ABB RobotStudio station: MiniProiect_v2final.rspag

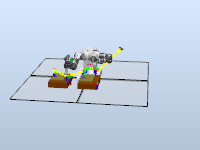
--- station ---
Station MiniProiect2 (saved by RobotStudio 7.0.8730.594)
Controller YuMi
  mechanical unit ROB_R: IRB14000_0.5_0.5_R, 6 joints, base frame (0, 0, 0) mm
  mechanical unit ROB_R_7: IRB14000_0.5_0.5_R, 1 joints, base frame (0, 0, 0) mm
  mechanical unit ROB_L: IRB14000_0.5_0.5_L, 6 joints, base frame (0, 0, 0) mm
  mechanical unit ROB_L_7: IRB14000_0.5_0.5_L, 1 joints, base frame (0, 0, 0) mm
Layout (positions relative to the parent item):
  - IRB14000_0.5_0.5 [mechanism, from Robots\IRB14000_0.5_0.5__01.rslib] at (0, 0, 0) mm
  - IRB14000_0.5_0.5_R [mechanism, from Robots\IRB14000_0.5_0.5__01.rslib] at (0, 0, 0) mm; joint values [2.2467, -1.1641, -0.2452, 0.0995, -2.8474, 1.8685, 0.012] (rad or m)
  - IRB14000_0.5_0.5_L [mechanism, from Robots\IRB14000_0.5_0.5__01.rslib] at (0, 0, 0) mm; joint values [-0.9882, -1.1775, 0.9709, 1.2171, -1.1721, -1.5184, 1.7927] (rad or m)
  - Curve_thing [part, from Training Objects\Curve_Thing.rslib] at (300, -50, 90) mm
  - Smart_Gripper_Servo_Fingers [mechanism, from Tools\ABB_Smart_Gripper_Servo_Fingers.rslib] at (305.45, 153.32, 394.2) mm, rotated rx 180 ry 0 rz 180 deg; joint values [0] (rad or m)
  - MyTool_2 [mechanism, from Training Objects\myTool.rslib] at (623.67, -200, 500.53) mm, rotated rx -180 ry 38 rz -180 deg
  - Curve [part, from Training Objects\Curve_Thing.rslib] at (300, -500, 90) mm
  - Part_3 [part] at (500.36, 1.06, 247.73) mm, rotated rx 179.59 ry 1.47 rz 162.83 deg
  - Part_4 [part] at (500, 0, 250) mm, rotated rx 180 ry 0 rz 84.95 deg
  - Attacher [smart component, from Components\Attacher.rslib]
      properties: Parent=MyTool_2; Flange=0; Child=Part_3; Mount=false; Offset=[0 0 0]; Orientation=[0 0 0]
  - Detacher [smart component, from Components\Detacher.rslib]
      properties: Child=Part_3; KeepPosition=true
  - CollisionSensor [smart component, from Components\CollisionSensor.rslib]
      properties: Object1=MyTool_2; Object2=Part_3; NearMiss=0.01; Part1=(none); Part2=(none); CollisionType=0
    - _sensorPart_ [part]
  - CollisionSensor_2 [smart component, from Components\CollisionSensor.rslib]
      properties: Object1=MyTool_2; Object2=Part_4; NearMiss=0.01; Part1=(none); Part2=(none); CollisionType=0
    - _sensorPart_ [part]
  - Positioner [smart component, from Components\Positioner.rslib]
      properties: Object=Part_3; Position=[0.477076 -0.45939 0.25]; Orientation=[0 0 0]; Reference=Global; ReferenceObject=(none)
Attachment: Smart_Gripper_Servo_Fingers is attached to IRB14000_0.5_0.5_L / Link7
Attachment: MyTool_2 is attached to IRB14000_0.5_0.5_R / Link7
Station signals: DI reset
Station logic (signal -> signal, property => property):
  MiniProiect2.reset -> Positioner.Execute
  CollisionSensor.SensorOut -> Attacher.Execute
  CollisionSensor_2.SensorOut -> Detacher.Execute

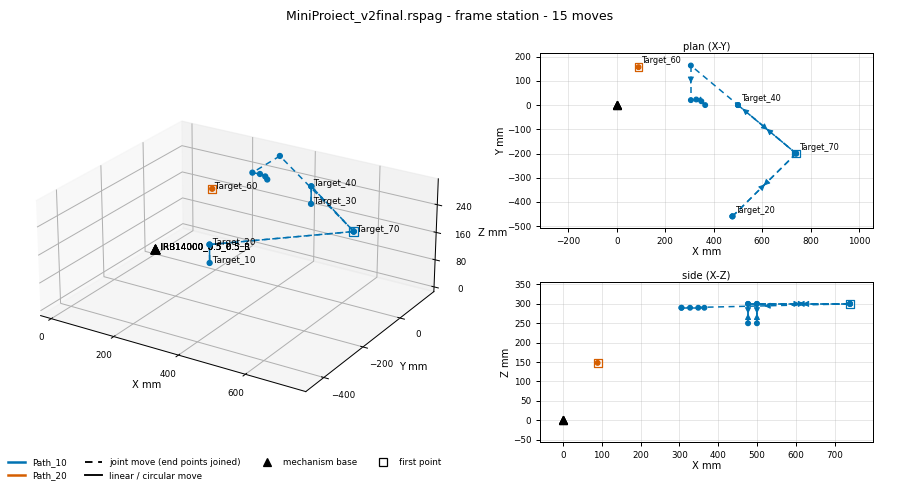
[picture p0: tool path of MiniProiect_v2final.rspag in frame station, 15 of 27 moves have a stored position in this frame; points joined in program order, loops and branches not executed]
--- Backups/YuMi/RAPID/TASK1/PROGMOD/CalibData.mod ---
MODULE CalibData
	PERS tooldata IRB5350_Gripper:=[TRUE,[[350,0,243],[0,1,0,0]],[1,[0,0,100],[1,0,0,0],0,0,0]];
	PERS tooldata MyTool:=[TRUE,[[31.7926,0,229.639],[0.945519,0,0.325568,0]],[1,[0,0,1],[1,0,0,0],0,0,0]];
ENDMODULE

--- Backups/YuMi/RAPID/TASK1/PROGMOD/Module1.mod ---
MODULE Module1
	CONST robtarget Target_70:=[[740,-200.004,300],[0,0,1,0],[1,-1,0,4],[-101.764306343,9E+09,9E+09,9E+09,9E+09,9E+09]];
	CONST robtarget Target_10:=[[477.07615446,-459.390112623,249.999908006],[-0.000000218,0.173648122,0.984807763,-0.000000081],[1,-2,0,4],[-101.764290321,9E+09,9E+09,9E+09,9E+09,9E+09]];
	CONST robtarget Target_20:=[[477.076,-459.39,300],[0,0.173648178,0.984807753,0],[1,-2,0,4],[-101.764306343,9E+09,9E+09,9E+09,9E+09,9E+09]];
	CONST robtarget Target_40:=[[500,0,300],[0,-0.173648177,0.984807753,0],[1,-2,0,4],[-101.764306343,9E+09,9E+09,9E+09,9E+09,9E+09]];
	CONST robtarget Target_30:=[[500,0,250],[0,-0.173648177,0.984807753,0],[1,-2,0,4],[-101.764306343,9E+09,9E+09,9E+09,9E+09,9E+09]];
    !***********************************************************
    !
    ! Module:  Module1
    !
    ! Description:
    !   <Insert description here>
    !
    ! Author: theod
    !
    ! Version: 1.0
    !
    !***********************************************************


    !***********************************************************
    !
    ! Procedure main
    !
    !   This is the entry point of your program
    !
    !***********************************************************
    PROC main()
        !Add your code here
    ENDPROC
	PROC Path_10()
	    MoveJ Target_70,v200,fine,MyTool\WObj:=wobj0;
	    MoveJ Target_20,v200,fine,MyTool\WObj:=wobj0;
	    MoveJ Target_10,v200,fine,MyTool\WObj:=wobj0;
	    MoveL Target_20,v1000,z100,MyTool\WObj:=wobj0;
	    MoveJ Target_70,v200,fine,MyTool\WObj:=wobj0;
	    MoveJ Target_40,v200,fine,MyTool\WObj:=wobj0;
	    MoveJ Target_30,v200,fine,MyTool\WObj:=wobj0;
	    MoveL Target_40,v1000,z100,MyTool\WObj:=wobj0;
	    MoveJ Target_70,v200,fine,MyTool\WObj:=wobj0;
	ENDPROC
ENDMODULE

--- Backups/YuMi/RAPID/TASK2/PROGMOD/CalibData.mod ---
MODULE CalibData
	PERS wobjdata Workobject_2:=[FALSE,TRUE,"",[[521.091,38.6689,180],[0,0.737574,0.675266,0]],[[0,0,0],[1,0,0,0]]];
	PERS wobjdata Workobject_3:=[FALSE,TRUE,"",[[477.076,-459.39,180],[0,0.737574,0.675266,0]],[[0,0,0],[1,0,0,0]]];
ENDMODULE

--- Backups/YuMi/RAPID/TASK2/PROGMOD/Module1.mod ---
MODULE Module1
	PERS tooldata Servo:=[TRUE,[[0,0,114.2],[1,0,0,0]],[0.215,[8.7,12.3,49.2],[1,0,0,0],0.00021,0.00024,0.00009]];
	PERS wobjdata Workobject_1:=[FALSE,TRUE,"",[[699.999,249.996,180],[0,-0.707107,0.707107,0]],[[0,0,0],[1,0,0,0]]];
	CONST robtarget Target_10:=[[86.674039551,394.552253174,-110],[0.707106781,0,0,0.707106781],[-1,-1,1,5],[135,9E+09,9E+09,9E+09,9E+09,9E+09]];
	CONST robtarget Target_20:=[[229.547583792,394.552253174,-110],[0.707106781,0,0,0.707106781],[-1,-1,1,5],[135,9E+09,9E+09,9E+09,9E+09,9E+09]];
	CONST robtarget Target_30:=[[226.937896068,372.374442925,-110],[0.707106781,0,0,0.707106781],[-1,-1,1,5],[135,9E+09,9E+09,9E+09,9E+09,9E+09]];
	CONST robtarget Target_40:=[[234.243334971,351.272398004,-110],[0.707106781,0,0,0.707106781],[-1,-1,1,5],[135,9E+09,9E+09,9E+09,9E+09,9E+09]];
	CONST robtarget Target_50:=[[250.00671167,335.455265126,-110],[0.707106781,0,0,0.707106781],[-1,-1,1,5],[135,9E+09,9E+09,9E+09,9E+09,9E+09]];
	CONST robtarget Target_60:=[[93.373882043,610.611053577,32.086529783],[0.674322362,0.323188765,0.416542029,-0.517040725],[0,0,0,4],[101.964427132,9E+09,9E+09,9E+09,9E+09,9E+09]];
	CONST jointtarget JointTarget_1:=[[-32.11,-102,-5.71,-103,-56.09,83.99],[0,9E+09,9E+09,9E+09,9E+09,9E+09]];
    CONST jointtarget JointTarget_2:=[[-32.11,-48.5,-5.71,-103,-56.09,83.99],[0,9E+09,9E+09,9E+09,9E+09,9E+09]];

    PROC main()
        !Path_Shake;
        userCommand;
    ENDPROC
	PROC Path_10()
	    MoveJ Target_10,v300,fine,Servo\WObj:=Workobject_1;
	    MoveJ Target_20,v300,fine,Servo\WObj:=Workobject_1;
	    MoveJ Target_30,v300,fine,Servo\WObj:=Workobject_1;
	    MoveJ Target_40,v300,fine,Servo\WObj:=Workobject_1;
	    MoveJ Target_50,v300,fine,Servo\WObj:=Workobject_1;
	ENDPROC
	PROC Path_20()
	    MoveJ Target_60,v300,fine,Servo\WObj:=Workobject_1;
	    MoveAbsJ JointTarget_1,v300,fine,Servo\WObj:=Workobject_1;
	ENDPROC

    PROC userCommand()
        VAR num valTranslare;
        CONST robtarget Target_70:=[[96.674039551,394.552253174,-110],[0.707106781,0,0,0.707106781],[-1,-1,1,5],[135,9E+09,9E+09,9E+09,9E+09,9E+09]];
        CONST robtarget Target_80:=[[126.674039551,394.552253174,-110],[0.707106781,0,0,0.707106781],[-1,-1,1,5],[135,9E+09,9E+09,9E+09,9E+09,9E+09]];
        CONST robtarget Target_90:=[[126.674039551,394.552253174,-90],[0.707106781,0,0,0.707106781],[-1,-1,1,5],[135,9E+09,9E+09,9E+09,9E+09,9E+09]];
        CONST robtarget Target_100:=[[96.674039551,394.552253174,-90],[0.707106781,0,0,0.707106781],[-1,-1,1,5],[135,9E+09,9E+09,9E+09,9E+09,9E+09]];
        TPReadNum valTranslare,"Dati o vloare pt translarea pe Z:";
        MoveJ RelTool(Target_10,0,0,valTranslare),v300,fine,Servo\WObj:=Workobject_1;
        WaitTime 2;
        MoveJ RelTool(Target_70,0,0,valTranslare),v300,fine,Servo\WObj:=Workobject_1;
        WaitTime 2;
        MoveJ RelTool(Target_80,0,0,valTranslare),v300,fine,Servo\WObj:=Workobject_1;
        WaitTime 2;
        MoveJ RelTool(Target_90,0,0,valTranslare),v300,fine,Servo\WObj:=Workobject_1;
        WaitTime 2;
        MoveJ RelTool(Target_100,0,0,valTranslare),v300,fine,Servo\WObj:=Workobject_1;
        WaitTime 2;
        MoveJ RelTool(Target_70,0,0,valTranslare),v300,fine,Servo\WObj:=Workobject_1;
    ENDPROC

    PROC Path_Shake()
        MoveAbsJ JointTarget_1,v300,fine,Servo\WObj:=Workobject_1;
        MoveAbsJ JointTarget_2,v300,fine,Servo\WObj:=Workobject_1;
        MoveAbsJ JointTarget_1,v300,fine,Servo\WObj:=Workobject_1;
        MoveAbsJ JointTarget_2,v300,fine,Servo\WObj:=Workobject_1;
        MoveAbsJ JointTarget_1,v300,fine,Servo\WObj:=Workobject_1;
    ENDPROC
ENDMODULE

--- Backups/YuMi/SYSPAR/EIO.cfg ---
EIO:CFG_1.0:6:1::
#
SYSSIG_IN:

      -Signal "Collision_Avoidance" -Action "CollAvoidance"
#
INDUSTRIAL_NETWORK:

      -Name "EtherNetIP" -Connection "Private Network"\
      -Label "EtherNet/IP Adapter Network"

      -Name "DeviceNet" -Label "DeviceNet Master/Slave Network" -Address "2"
#
EIO_CROSS:

      -Name "Cross_Signal_Lamp" -Res "Signal_Lamp" -Act1 "DRV1BRAKE"
#
EIO_SIGNAL_SAFELEVEL:

      -Name "FlangePowerSafeLevel" -ActionWhenStartup "Last"
#
DEVICENET_DEVICE:

      -Name "D652_10" -VendorName "ABB Robotics" -ProductName "24 VDC Unit"\
      -Address 10 -ProductCode 26 -DeviceType 7 -ConnectionType "COS"\
      -OutputSize 2 -InputSize 2
#
DEVICENET_INTERNAL_DEVICE:

      -Name "DN_Internal_Device" -VendorName "ABB Robotics"\
      -ProductName "DeviceNet Internal Slave Device"
#
ETHERNETIP_INTERNAL_DEVICE:

      -Name "EN_Internal_Device" -VendorName "ABB Robotics"\
      -ProductName "EtherNet/IP Internal Adapter Device"
#
EIO_SIGNAL:

      -Name "custom_DI_0" -SignalType "DI" -Device "D652_10" -DeviceMap "0"

      -Name "custom_DI_1" -SignalType "DI" -Device "D652_10" -DeviceMap "1"

      -Name "custom_DI_2" -SignalType "DI" -Device "D652_10" -DeviceMap "2"

      -Name "custom_DI_3" -SignalType "DI" -Device "D652_10" -DeviceMap "3"

      -Name "custom_DI_4" -SignalType "DI" -Device "D652_10" -DeviceMap "4"

      -Name "custom_DI_5" -SignalType "DI" -Device "D652_10" -DeviceMap "5"

      -Name "custom_DI_6" -SignalType "DI" -Device "D652_10" -DeviceMap "6"

      -Name "custom_DI_7" -SignalType "DI" -Device "D652_10" -DeviceMap "7"

      -Name "custom_DO_0" -SignalType "DO" -Device "D652_10" -DeviceMap "0"

      -Name "custom_DO_1" -SignalType "DO" -Device "D652_10" -DeviceMap "1"

      -Name "custom_DO_2" -SignalType "DO" -Device "D652_10" -DeviceMap "2"

      -Name "custom_DO_3" -SignalType "DO" -Device "D652_10" -DeviceMap "3"

      -Name "custom_DO_4" -SignalType "DO" -Device "D652_10" -DeviceMap "4"

      -Name "custom_DO_5" -SignalType "DO" -Device "D652_10" -DeviceMap "5"

      -Name "custom_DO_6" -SignalType "DO" -Device "D652_10" -DeviceMap "6"

      -Name "custom_DO_7" -SignalType "DO" -Device "D652_10" -DeviceMap "7"

      -Name "hall_sensor_joint_1" -SignalType "DI" -Device "D652_10"\
      -DeviceMap "8"

      -Name "hall_sensor_joint_2" -SignalType "DI" -Device "D652_10"\
      -DeviceMap "9"

      -Name "hall_sensor_joint_3" -SignalType "DI" -Device "D652_10"\
      -DeviceMap "11"

      -Name "hall_sensor_joint_4" -SignalType "DI" -Device "D652_10"\
      -DeviceMap "12"

      -Name "hall_sensor_joint_5" -SignalType "DI" -Device "D652_10"\
      -DeviceMap "13"

      -Name "hall_sensor_joint_6" -SignalType "DI" -Device "D652_10"\
      -DeviceMap "14"

      -Name "hall_sensor_joint_7" -SignalType "DI" -Device "D652_10"\
      -DeviceMap "10"

      -Name "hall_sensor_24V_ROB_R" -SignalType "DO" -Device "D652_10"\
      -DeviceMap "8"

      -Name "hall_sensor_24V_ROB_L" -SignalType "DO" -Device "D652_10"\
      -DeviceMap "9"

      -Name "flange_24V_ROB_R" -SignalType "DO" -Device "D652_10"\
      -DeviceMap "10" -SafeLevel "FlangePowerSafeLevel"

      -Name "flange_24V_ROB_L" -SignalType "DO" -Device "D652_10"\
      -DeviceMap "11" -SafeLevel "FlangePowerSafeLevel"

      -Name "Signal_Lamp" -SignalType "DO" -Device "D652_10" -DeviceMap "12"

      -Name "Collision_Avoidance" -SignalType "DO" -Access "All" -Default 1
